ABB RAPID module: RRC_DataGlobal_Ctrl.sysx

MODULE RRC_DataGlobal_Ctrl(SYSMODULE)
    !***********************************************************************************
    !
    ! ETH Zurich / Robotic Fabrication Lab
    ! HIB C13 / Stefano-Franscini-Platz 1
    ! CH-8093 Zurich
    !
    !***********************************************************************************
    !
    ! PROJECT     :  RRC - Rapid Robot Communication
    !
    ! FUNCTION    :  Inclouds all project spezific global datas
    !
    ! AUTHOR      :  Philippe Fleischmann
    !
    ! EMAIL       :  rrc@arch.ethz.ch
    !
    ! HISTORY     :  2019.02.22
    !
    ! Copyright   :  ETH Zurich (CH) 2019
    !                - Philippe Fleischmann
    !                - Michael Lyrenmann
    !                - Gonzalo Casas
    !
    ! License     :  This code base is governed by an EULA (End-User License Agreement)
    !                which you have received together with the software.
    !                You are not allowed to use the software on a real robots
    !                without a signed EULA.
    !
    !                A copy of the EULA content is in the controller task (T_CTRL).
    !
    !***********************************************************************************

    !************************************************
    ! Declaration :     bool
    !************************************************
    !
    PERS bool b_RRC_TaskReceiverOn:=TRUE;
    PERS bool b_RRC_TaskSenderOn:=TRUE;
    !
    PERS bool b_RRC_CtrlWaitForJob:=TRUE;
    PERS bool b_RRC_CtrlHamModOn:=FALSE;
    PERS bool b_RRC_CtrlInUse:=FALSE;
    PERS bool b_RRC_AutoIPAddress:=FALSE;
    PERS bool b_RRC_VirtualCustomPorts:=FALSE;
    !
    ! Channels
    PERS bool b_RRC_Com{n_RRC_NumOfCha}:=[TRUE,FALSE,FALSE,FALSE];
    PERS bool b_RRC_SIDCheck{n_RRC_NumOfCha}:=[TRUE,FALSE,FALSE,FALSE];
    PERS bool b_RRC_SIDErrorStop{n_RRC_NumOfCha}:=[FALSE,FALSE,FALSE,FALSE];
    PERS bool b_RRC_LogPro{n_RRC_NumOfCha}:=[FALSE,FALSE,FALSE,FALSE];
    !
    ! Client information
    PERS bool b_RRC_PPMain:=TRUE;
    !
    ! Activate or deactivate a event log message
    PERS bool b_RRC_EvLogReadAndUnpackTime:=FALSE;
    PERS bool b_RRC_EvLogPackAndSendTime:=FALSE;
    PERS bool b_RRC_EvLogMsgInUntilMsgOutTime:=FALSE;
    !
    ! Temporary to measure the feedback loop
    PERS bool b_RRC_FeedbackOut:=TRUE;

    !************************************************
    ! Declaration :     num
    !************************************************
    !
    !* PERS num n_RRC_WritePtrSenBufRob1:=1;
    PERS num n_RRC_WritePtrSenBufCtrl{n_RRC_NumOfCha}:=[0,0,0,0];
    PERS num n_RRC_WritePtrSenBufRob{n_RRC_NumOfCha}:=[4,0,0,0];
    !* PERS num n_RRC_SIDMax:=8388608;
    PERS num n_RRC_SIDMax:=1000000;
    !
    PERS num n_RRC_R1_ChaNr:=1;
    PERS num n_RRC_R2_ChaNr:=2;
    PERS num n_RRC_R3_ChaNr:=3;
    PERS num n_RRC_R4_ChaNr:=4;
    !
    PERS num n_RRC_SocketPortRec{n_RRC_NumOfCha}:=[30101,30102,30103,30104];
    PERS num n_RRC_SocketPortSen{n_RRC_NumOfCha}:=[30201,30202,30203,30204];
    !
    PERS num n_RRC_TimeTaskLiAll:=0.1;
    PERS num n_RRC_TimeTPMsg:=0.5;
    !
    PERS num n_RRC_ProtocolVersion:=2;

    !************************************************
    ! Declaration :     string
    !************************************************
    !
    PERS string n_RRC_Version:="v1.1.0";
    !
    PERS string st_RRC_CurCtrlJob:="RRC";
    PERS string st_RRC_JobForCtrl:="r_A031_HamMod";
    !
    PERS string st_RRC_IP_Address:="192.168.125.1";
    PERS string st_RRC_IP_AddressVC:="127.0.0.1";
    PERS string st_RRC_IP_AddressMan:="192.168.125.1";
    !
    ! System data
    PERS string st_RRC_SerialNr:="15000-100220";
    PERS string st_RRC_SoftwareVersion:="7.7.1+296";
    PERS string st_RRC_RobotWare:="7.7.1";
    PERS string st_RRC_ControllerID:="15000-100220";
    PERS string st_RRC_WAN_IP:="0.0.0.0";
    PERS string st_RRC_ControllerLang:="en";
    PERS string st_RRC_SystemName:="15000-100220";

    !************************************************
    ! Declaration :     tasklist
    !************************************************
    !
    PERS tasks tl_RRC_All{7}:=[["T_CTRL"],["T_RX"],["T_TX"],["T_ROB1"],[""],[""],[""]];

    !************************************************
    ! Declaration :     syncident
    !************************************************
    !
    VAR syncident id_RRC_MainSta;
    VAR syncident id_RRC_MainEnd;
    !
    VAR syncident id_RRC_InitSta;
    VAR syncident id_RRC_InitCtrl;
    VAR syncident id_RRC_InitEnd;

    !************************************************
    ! Declaration :     RRC_Channel
    !************************************************
    !
    PERS RRC_Channel ch_RRC_Channels:=[["T_ROB1",1],["T_ROB2",2],["T_ROB3",3],["T_ROB4",4]];

    !************************************************
    ! Declaration :     RRC_buffer_msg
    !************************************************
    !
    ! Receiver buffer for controller
    PERS RRC_buffer_msg bm_RRC_RecBufferCtrl{n_RRC_NumOfCha,10}:=[
    [[[0,0,0,"",0,0,"",0,0,0,"",0,"",0,"",0,"",0,"",0,"",0,"",0,"",0,0,0,0,0,0,0,0,0,0,0,0,0,0,0,0,0,0,0,0,0,0,0,0,0,0,0,0,0,0,0,0,0,0,0,0,0],FALSE],
    [[0,0,0,"",0,0,"",0,0,0,"",0,"",0,"",0,"",0,"",0,"",0,"",0,"",0,0,0,0,0,0,0,0,0,0,0,0,0,0,0,0,0,0,0,0,0,0,0,0,0,0,0,0,0,0,0,0,0,0,0,0,0],FALSE],
    [[0,0,0,"",0,0,"",0,0,0,"",0,"",0,"",0,"",0,"",0,"",0,"",0,"",0,0,0,0,0,0,0,0,0,0,0,0,0,0,0,0,0,0,0,0,0,0,0,0,0,0,0,0,0,0,0,0,0,0,0,0,0],FALSE],
    [[0,0,0,"",0,0,"",0,0,0,"",0,"",0,"",0,"",0,"",0,"",0,"",0,"",0,0,0,0,0,0,0,0,0,0,0,0,0,0,0,0,0,0,0,0,0,0,0,0,0,0,0,0,0,0,0,0,0,0,0,0,0],FALSE],
    [[0,0,0,"",0,0,"",0,0,0,"",0,"",0,"",0,"",0,"",0,"",0,"",0,"",0,0,0,0,0,0,0,0,0,0,0,0,0,0,0,0,0,0,0,0,0,0,0,0,0,0,0,0,0,0,0,0,0,0,0,0,0],FALSE],
    [[0,0,0,"",0,0,"",0,0,0,"",0,"",0,"",0,"",0,"",0,"",0,"",0,"",0,0,0,0,0,0,0,0,0,0,0,0,0,0,0,0,0,0,0,0,0,0,0,0,0,0,0,0,0,0,0,0,0,0,0,0,0],FALSE],
    [[0,0,0,"",0,0,"",0,0,0,"",0,"",0,"",0,"",0,"",0,"",0,"",0,"",0,0,0,0,0,0,0,0,0,0,0,0,0,0,0,0,0,0,0,0,0,0,0,0,0,0,0,0,0,0,0,0,0,0,0,0,0],FALSE],
    [[0,0,0,"",0,0,"",0,0,0,"",0,"",0,"",0,"",0,"",0,"",0,"",0,"",0,0,0,0,0,0,0,0,0,0,0,0,0,0,0,0,0,0,0,0,0,0,0,0,0,0,0,0,0,0,0,0,0,0,0,0,0],FALSE],
    [[0,0,0,"",0,0,"",0,0,0,"",0,"",0,"",0,"",0,"",0,"",0,"",0,"",0,0,0,0,0,0,0,0,0,0,0,0,0,0,0,0,0,0,0,0,0,0,0,0,0,0,0,0,0,0,0,0,0,0,0,0,0],FALSE],
    [[0,0,0,"",0,0,"",0,0,0,"",0,"",0,"",0,"",0,"",0,"",0,"",0,"",0,0,0,0,0,0,0,0,0,0,0,0,0,0,0,0,0,0,0,0,0,0,0,0,0,0,0,0,0,0,0,0,0,0,0,0,0],FALSE]],

    [[[0,0,0,"",0,0,"",0,0,0,"",0,"",0,"",0,"",0,"",0,"",0,"",0,"",0,0,0,0,0,0,0,0,0,0,0,0,0,0,0,0,0,0,0,0,0,0,0,0,0,0,0,0,0,0,0,0,0,0,0,0,0],FALSE],
    [[0,0,0,"",0,0,"",0,0,0,"",0,"",0,"",0,"",0,"",0,"",0,"",0,"",0,0,0,0,0,0,0,0,0,0,0,0,0,0,0,0,0,0,0,0,0,0,0,0,0,0,0,0,0,0,0,0,0,0,0,0,0],FALSE],
    [[0,0,0,"",0,0,"",0,0,0,"",0,"",0,"",0,"",0,"",0,"",0,"",0,"",0,0,0,0,0,0,0,0,0,0,0,0,0,0,0,0,0,0,0,0,0,0,0,0,0,0,0,0,0,0,0,0,0,0,0,0,0],FALSE],
    [[0,0,0,"",0,0,"",0,0,0,"",0,"",0,"",0,"",0,"",0,"",0,"",0,"",0,0,0,0,0,0,0,0,0,0,0,0,0,0,0,0,0,0,0,0,0,0,0,0,0,0,0,0,0,0,0,0,0,0,0,0,0],FALSE],
    [[0,0,0,"",0,0,"",0,0,0,"",0,"",0,"",0,"",0,"",0,"",0,"",0,"",0,0,0,0,0,0,0,0,0,0,0,0,0,0,0,0,0,0,0,0,0,0,0,0,0,0,0,0,0,0,0,0,0,0,0,0,0],FALSE],
    [[0,0,0,"",0,0,"",0,0,0,"",0,"",0,"",0,"",0,"",0,"",0,"",0,"",0,0,0,0,0,0,0,0,0,0,0,0,0,0,0,0,0,0,0,0,0,0,0,0,0,0,0,0,0,0,0,0,0,0,0,0,0],FALSE],
    [[0,0,0,"",0,0,"",0,0,0,"",0,"",0,"",0,"",0,"",0,"",0,"",0,"",0,0,0,0,0,0,0,0,0,0,0,0,0,0,0,0,0,0,0,0,0,0,0,0,0,0,0,0,0,0,0,0,0,0,0,0,0],FALSE],
    [[0,0,0,"",0,0,"",0,0,0,"",0,"",0,"",0,"",0,"",0,"",0,"",0,"",0,0,0,0,0,0,0,0,0,0,0,0,0,0,0,0,0,0,0,0,0,0,0,0,0,0,0,0,0,0,0,0,0,0,0,0,0],FALSE],
    [[0,0,0,"",0,0,"",0,0,0,"",0,"",0,"",0,"",0,"",0,"",0,"",0,"",0,0,0,0,0,0,0,0,0,0,0,0,0,0,0,0,0,0,0,0,0,0,0,0,0,0,0,0,0,0,0,0,0,0,0,0,0],FALSE],
    [[0,0,0,"",0,0,"",0,0,0,"",0,"",0,"",0,"",0,"",0,"",0,"",0,"",0,0,0,0,0,0,0,0,0,0,0,0,0,0,0,0,0,0,0,0,0,0,0,0,0,0,0,0,0,0,0,0,0,0,0,0,0],FALSE]],

    [[[0,0,0,"",0,0,"",0,0,0,"",0,"",0,"",0,"",0,"",0,"",0,"",0,"",0,0,0,0,0,0,0,0,0,0,0,0,0,0,0,0,0,0,0,0,0,0,0,0,0,0,0,0,0,0,0,0,0,0,0,0,0],FALSE],
    [[0,0,0,"",0,0,"",0,0,0,"",0,"",0,"",0,"",0,"",0,"",0,"",0,"",0,0,0,0,0,0,0,0,0,0,0,0,0,0,0,0,0,0,0,0,0,0,0,0,0,0,0,0,0,0,0,0,0,0,0,0,0],FALSE],
    [[0,0,0,"",0,0,"",0,0,0,"",0,"",0,"",0,"",0,"",0,"",0,"",0,"",0,0,0,0,0,0,0,0,0,0,0,0,0,0,0,0,0,0,0,0,0,0,0,0,0,0,0,0,0,0,0,0,0,0,0,0,0],FALSE],
    [[0,0,0,"",0,0,"",0,0,0,"",0,"",0,"",0,"",0,"",0,"",0,"",0,"",0,0,0,0,0,0,0,0,0,0,0,0,0,0,0,0,0,0,0,0,0,0,0,0,0,0,0,0,0,0,0,0,0,0,0,0,0],FALSE],
    [[0,0,0,"",0,0,"",0,0,0,"",0,"",0,"",0,"",0,"",0,"",0,"",0,"",0,0,0,0,0,0,0,0,0,0,0,0,0,0,0,0,0,0,0,0,0,0,0,0,0,0,0,0,0,0,0,0,0,0,0,0,0],FALSE],
    [[0,0,0,"",0,0,"",0,0,0,"",0,"",0,"",0,"",0,"",0,"",0,"",0,"",0,0,0,0,0,0,0,0,0,0,0,0,0,0,0,0,0,0,0,0,0,0,0,0,0,0,0,0,0,0,0,0,0,0,0,0,0],FALSE],
    [[0,0,0,"",0,0,"",0,0,0,"",0,"",0,"",0,"",0,"",0,"",0,"",0,"",0,0,0,0,0,0,0,0,0,0,0,0,0,0,0,0,0,0,0,0,0,0,0,0,0,0,0,0,0,0,0,0,0,0,0,0,0],FALSE],
    [[0,0,0,"",0,0,"",0,0,0,"",0,"",0,"",0,"",0,"",0,"",0,"",0,"",0,0,0,0,0,0,0,0,0,0,0,0,0,0,0,0,0,0,0,0,0,0,0,0,0,0,0,0,0,0,0,0,0,0,0,0,0],FALSE],
    [[0,0,0,"",0,0,"",0,0,0,"",0,"",0,"",0,"",0,"",0,"",0,"",0,"",0,0,0,0,0,0,0,0,0,0,0,0,0,0,0,0,0,0,0,0,0,0,0,0,0,0,0,0,0,0,0,0,0,0,0,0,0],FALSE],
    [[0,0,0,"",0,0,"",0,0,0,"",0,"",0,"",0,"",0,"",0,"",0,"",0,"",0,0,0,0,0,0,0,0,0,0,0,0,0,0,0,0,0,0,0,0,0,0,0,0,0,0,0,0,0,0,0,0,0,0,0,0,0],FALSE]],

    [[[0,0,0,"",0,0,"",0,0,0,"",0,"",0,"",0,"",0,"",0,"",0,"",0,"",0,0,0,0,0,0,0,0,0,0,0,0,0,0,0,0,0,0,0,0,0,0,0,0,0,0,0,0,0,0,0,0,0,0,0,0,0],FALSE],
    [[0,0,0,"",0,0,"",0,0,0,"",0,"",0,"",0,"",0,"",0,"",0,"",0,"",0,0,0,0,0,0,0,0,0,0,0,0,0,0,0,0,0,0,0,0,0,0,0,0,0,0,0,0,0,0,0,0,0,0,0,0,0],FALSE],
    [[0,0,0,"",0,0,"",0,0,0,"",0,"",0,"",0,"",0,"",0,"",0,"",0,"",0,0,0,0,0,0,0,0,0,0,0,0,0,0,0,0,0,0,0,0,0,0,0,0,0,0,0,0,0,0,0,0,0,0,0,0,0],FALSE],
    [[0,0,0,"",0,0,"",0,0,0,"",0,"",0,"",0,"",0,"",0,"",0,"",0,"",0,0,0,0,0,0,0,0,0,0,0,0,0,0,0,0,0,0,0,0,0,0,0,0,0,0,0,0,0,0,0,0,0,0,0,0,0],FALSE],
    [[0,0,0,"",0,0,"",0,0,0,"",0,"",0,"",0,"",0,"",0,"",0,"",0,"",0,0,0,0,0,0,0,0,0,0,0,0,0,0,0,0,0,0,0,0,0,0,0,0,0,0,0,0,0,0,0,0,0,0,0,0,0],FALSE],
    [[0,0,0,"",0,0,"",0,0,0,"",0,"",0,"",0,"",0,"",0,"",0,"",0,"",0,0,0,0,0,0,0,0,0,0,0,0,0,0,0,0,0,0,0,0,0,0,0,0,0,0,0,0,0,0,0,0,0,0,0,0,0],FALSE],
    [[0,0,0,"",0,0,"",0,0,0,"",0,"",0,"",0,"",0,"",0,"",0,"",0,"",0,0,0,0,0,0,0,0,0,0,0,0,0,0,0,0,0,0,0,0,0,0,0,0,0,0,0,0,0,0,0,0,0,0,0,0,0],FALSE],
    [[0,0,0,"",0,0,"",0,0,0,"",0,"",0,"",0,"",0,"",0,"",0,"",0,"",0,0,0,0,0,0,0,0,0,0,0,0,0,0,0,0,0,0,0,0,0,0,0,0,0,0,0,0,0,0,0,0,0,0,0,0,0],FALSE],
    [[0,0,0,"",0,0,"",0,0,0,"",0,"",0,"",0,"",0,"",0,"",0,"",0,"",0,0,0,0,0,0,0,0,0,0,0,0,0,0,0,0,0,0,0,0,0,0,0,0,0,0,0,0,0,0,0,0,0,0,0,0,0],FALSE],
    [[0,0,0,"",0,0,"",0,0,0,"",0,"",0,"",0,"",0,"",0,"",0,"",0,"",0,0,0,0,0,0,0,0,0,0,0,0,0,0,0,0,0,0,0,0,0,0,0,0,0,0,0,0,0,0,0,0,0,0,0,0,0],FALSE]]];

    !
    ! Receiver buffer for robots
    PERS RRC_buffer_msg bm_RRC_RecBufferRob{n_RRC_NumOfCha,10}:=[
    [[[5,0,12,"r_RRC_MoveTo",1,0,"",0,1,6,"FrameL",0,"",0,"",0,"",0,"",0,"",0,"",0,"",15,0.00865957,478.991,218.552,7.09225E-05,0.923882,-0.382677,3.67571E-05,0,0,0,0,0,0,300,-1,0,0,0,0,0,0,0,0,0,0,0,0,0,0,0,0,0,0,0,0,0],FALSE],
    [[6,0,12,"r_RRC_MoveTo",1,0,"",0,1,6,"FrameL",0,"",0,"",0,"",0,"",0,"",0,"",0,"",15,550.001,-0.000425997,717.995,-1.78564E-06,-0.382682,0.92388,7.29413E-07,0,0,0,0,0,0,300,-1,0,0,0,0,0,0,0,0,0,0,0,0,0,0,0,0,0,0,0,0,0],FALSE],
    [[7,0,12,"r_RRC_MoveTo",1,0,"",0,1,6,"FrameL",0,"",0,"",0,"",0,"",0,"",0,"",0,"",15,697.669,-21.8245,303.5,0,-0.320157,0.947365,0,0,0,0,0,0,0,300,-1,0,0,0,0,0,0,0,0,0,0,0,0,0,0,0,0,0,0,0,0,0],FALSE],
    [[8,0,12,"r_RRC_MoveTo",1,0,"",0,1,6,"FrameL",0,"",0,"",0,"",0,"",0,"",0,"",0,"",15,697.669,-21.8245,253.5,0,-0.320157,0.947365,0,0,0,0,0,0,0,300,-1,0,0,0,0,0,0,0,0,0,0,0,0,0,0,0,0,0,0,0,0,0],FALSE],
    [[9,0,16,"r_RRC_SetDigital",0,0,"",0,1,22,"ABB_Scalable_IO_0_DO16",0,"",0,"",0,"",0,"",0,"",0,"",0,"",1,1,-21.8245,253.5,0,-0.320157,0.947365,0,0,0,0,0,0,0,300,-1,0,0,0,0,0,0,0,0,0,0,0,0,0,0,0,0,0,0,0,0,0],FALSE],
    [[10,0,12,"r_RRC_MoveTo",1,0,"",0,1,6,"FrameL",0,"",0,"",0,"",0,"",0,"",0,"",0,"",15,697.669,-21.8245,303.5,0,-0.320157,0.947365,0,0,0,0,0,0,0,300,-1,0,0,0,0,0,0,0,0,0,0,0,0,0,0,0,0,0,0,0,0,0],FALSE],
    [[11,0,12,"r_RRC_MoveTo",1,0,"",0,1,6,"FrameL",0,"",0,"",0,"",0,"",0,"",0,"",0,"",15,550.001,-0.000425997,717.995,-1.78564E-06,-0.382682,0.92388,7.29413E-07,0,0,0,0,0,0,300,-1,0,0,0,0,0,0,0,0,0,0,0,0,0,0,0,0,0,0,0,0,0],FALSE],
    [[12,0,12,"r_RRC_MoveTo",1,0,"",0,1,6,"FrameL",0,"",0,"",0,"",0,"",0,"",0,"",0,"",15,0.00865957,478.991,218.552,7.09225E-05,0.923882,-0.382677,3.67571E-05,0,0,0,0,0,0,300,-1,0,0,0,0,0,0,0,0,0,0,0,0,0,0,0,0,0,0,0,0,0],FALSE],
    [[13,0,12,"r_RRC_MoveTo",1,0,"",0,1,6,"FrameL",0,"",0,"",0,"",0,"",0,"",0,"",0,"",15,0.00865957,478.991,168.552,7.09225E-05,0.923882,-0.382677,3.67571E-05,0,0,0,0,0,0,300,-1,0,0,0,0,0,0,0,0,0,0,0,0,0,0,0,0,0,0,0,0,0],FALSE],
    [[4,0,14,"r_RRC_WaitTime",1,0,"",0,0,22,"ABB_Scalable_IO_0_DO16",0,"",0,"",0,"",0,"",0,"",0,"",0,"",1,1,478.991,168.552,7.09225E-05,0.923882,-0.382677,3.67571E-05,0,0,0,0,0,0,300,-1,0,0,0,0,0,0,0,0,0,0,0,0,0,0,0,0,0,0,0,0,0],FALSE]],

    [[[0,0,0,"",0,0,"",0,0,0,"",0,"",0,"",0,"",0,"",0,"",0,"",0,"",0,0,0,0,0,0,0,0,0,0,0,0,0,0,0,0,0,0,0,0,0,0,0,0,0,0,0,0,0,0,0,0,0,0,0,0,0],FALSE],
    [[0,0,0,"",0,0,"",0,0,0,"",0,"",0,"",0,"",0,"",0,"",0,"",0,"",0,0,0,0,0,0,0,0,0,0,0,0,0,0,0,0,0,0,0,0,0,0,0,0,0,0,0,0,0,0,0,0,0,0,0,0,0],FALSE],
    [[0,0,0,"",0,0,"",0,0,0,"",0,"",0,"",0,"",0,"",0,"",0,"",0,"",0,0,0,0,0,0,0,0,0,0,0,0,0,0,0,0,0,0,0,0,0,0,0,0,0,0,0,0,0,0,0,0,0,0,0,0,0],FALSE],
    [[0,0,0,"",0,0,"",0,0,0,"",0,"",0,"",0,"",0,"",0,"",0,"",0,"",0,0,0,0,0,0,0,0,0,0,0,0,0,0,0,0,0,0,0,0,0,0,0,0,0,0,0,0,0,0,0,0,0,0,0,0,0],FALSE],
    [[0,0,0,"",0,0,"",0,0,0,"",0,"",0,"",0,"",0,"",0,"",0,"",0,"",0,0,0,0,0,0,0,0,0,0,0,0,0,0,0,0,0,0,0,0,0,0,0,0,0,0,0,0,0,0,0,0,0,0,0,0,0],FALSE],
    [[0,0,0,"",0,0,"",0,0,0,"",0,"",0,"",0,"",0,"",0,"",0,"",0,"",0,0,0,0,0,0,0,0,0,0,0,0,0,0,0,0,0,0,0,0,0,0,0,0,0,0,0,0,0,0,0,0,0,0,0,0,0],FALSE],
    [[0,0,0,"",0,0,"",0,0,0,"",0,"",0,"",0,"",0,"",0,"",0,"",0,"",0,0,0,0,0,0,0,0,0,0,0,0,0,0,0,0,0,0,0,0,0,0,0,0,0,0,0,0,0,0,0,0,0,0,0,0,0],FALSE],
    [[0,0,0,"",0,0,"",0,0,0,"",0,"",0,"",0,"",0,"",0,"",0,"",0,"",0,0,0,0,0,0,0,0,0,0,0,0,0,0,0,0,0,0,0,0,0,0,0,0,0,0,0,0,0,0,0,0,0,0,0,0,0],FALSE],
    [[0,0,0,"",0,0,"",0,0,0,"",0,"",0,"",0,"",0,"",0,"",0,"",0,"",0,0,0,0,0,0,0,0,0,0,0,0,0,0,0,0,0,0,0,0,0,0,0,0,0,0,0,0,0,0,0,0,0,0,0,0,0],FALSE],
    [[0,0,0,"",0,0,"",0,0,0,"",0,"",0,"",0,"",0,"",0,"",0,"",0,"",0,0,0,0,0,0,0,0,0,0,0,0,0,0,0,0,0,0,0,0,0,0,0,0,0,0,0,0,0,0,0,0,0,0,0,0,0],FALSE]],

    [[[0,0,0,"",0,0,"",0,0,0,"",0,"",0,"",0,"",0,"",0,"",0,"",0,"",0,0,0,0,0,0,0,0,0,0,0,0,0,0,0,0,0,0,0,0,0,0,0,0,0,0,0,0,0,0,0,0,0,0,0,0,0],FALSE],
    [[0,0,0,"",0,0,"",0,0,0,"",0,"",0,"",0,"",0,"",0,"",0,"",0,"",0,0,0,0,0,0,0,0,0,0,0,0,0,0,0,0,0,0,0,0,0,0,0,0,0,0,0,0,0,0,0,0,0,0,0,0,0],FALSE],
    [[0,0,0,"",0,0,"",0,0,0,"",0,"",0,"",0,"",0,"",0,"",0,"",0,"",0,0,0,0,0,0,0,0,0,0,0,0,0,0,0,0,0,0,0,0,0,0,0,0,0,0,0,0,0,0,0,0,0,0,0,0,0],FALSE],
    [[0,0,0,"",0,0,"",0,0,0,"",0,"",0,"",0,"",0,"",0,"",0,"",0,"",0,0,0,0,0,0,0,0,0,0,0,0,0,0,0,0,0,0,0,0,0,0,0,0,0,0,0,0,0,0,0,0,0,0,0,0,0],FALSE],
    [[0,0,0,"",0,0,"",0,0,0,"",0,"",0,"",0,"",0,"",0,"",0,"",0,"",0,0,0,0,0,0,0,0,0,0,0,0,0,0,0,0,0,0,0,0,0,0,0,0,0,0,0,0,0,0,0,0,0,0,0,0,0],FALSE],
    [[0,0,0,"",0,0,"",0,0,0,"",0,"",0,"",0,"",0,"",0,"",0,"",0,"",0,0,0,0,0,0,0,0,0,0,0,0,0,0,0,0,0,0,0,0,0,0,0,0,0,0,0,0,0,0,0,0,0,0,0,0,0],FALSE],
    [[0,0,0,"",0,0,"",0,0,0,"",0,"",0,"",0,"",0,"",0,"",0,"",0,"",0,0,0,0,0,0,0,0,0,0,0,0,0,0,0,0,0,0,0,0,0,0,0,0,0,0,0,0,0,0,0,0,0,0,0,0,0],FALSE],
    [[0,0,0,"",0,0,"",0,0,0,"",0,"",0,"",0,"",0,"",0,"",0,"",0,"",0,0,0,0,0,0,0,0,0,0,0,0,0,0,0,0,0,0,0,0,0,0,0,0,0,0,0,0,0,0,0,0,0,0,0,0,0],FALSE],
    [[0,0,0,"",0,0,"",0,0,0,"",0,"",0,"",0,"",0,"",0,"",0,"",0,"",0,0,0,0,0,0,0,0,0,0,0,0,0,0,0,0,0,0,0,0,0,0,0,0,0,0,0,0,0,0,0,0,0,0,0,0,0],FALSE],
    [[0,0,0,"",0,0,"",0,0,0,"",0,"",0,"",0,"",0,"",0,"",0,"",0,"",0,0,0,0,0,0,0,0,0,0,0,0,0,0,0,0,0,0,0,0,0,0,0,0,0,0,0,0,0,0,0,0,0,0,0,0,0],FALSE]],

    [[[0,0,0,"",0,0,"",0,0,0,"",0,"",0,"",0,"",0,"",0,"",0,"",0,"",0,0,0,0,0,0,0,0,0,0,0,0,0,0,0,0,0,0,0,0,0,0,0,0,0,0,0,0,0,0,0,0,0,0,0,0,0],FALSE],
    [[0,0,0,"",0,0,"",0,0,0,"",0,"",0,"",0,"",0,"",0,"",0,"",0,"",0,0,0,0,0,0,0,0,0,0,0,0,0,0,0,0,0,0,0,0,0,0,0,0,0,0,0,0,0,0,0,0,0,0,0,0,0],FALSE],
    [[0,0,0,"",0,0,"",0,0,0,"",0,"",0,"",0,"",0,"",0,"",0,"",0,"",0,0,0,0,0,0,0,0,0,0,0,0,0,0,0,0,0,0,0,0,0,0,0,0,0,0,0,0,0,0,0,0,0,0,0,0,0],FALSE],
    [[0,0,0,"",0,0,"",0,0,0,"",0,"",0,"",0,"",0,"",0,"",0,"",0,"",0,0,0,0,0,0,0,0,0,0,0,0,0,0,0,0,0,0,0,0,0,0,0,0,0,0,0,0,0,0,0,0,0,0,0,0,0],FALSE],
    [[0,0,0,"",0,0,"",0,0,0,"",0,"",0,"",0,"",0,"",0,"",0,"",0,"",0,0,0,0,0,0,0,0,0,0,0,0,0,0,0,0,0,0,0,0,0,0,0,0,0,0,0,0,0,0,0,0,0,0,0,0,0],FALSE],
    [[0,0,0,"",0,0,"",0,0,0,"",0,"",0,"",0,"",0,"",0,"",0,"",0,"",0,0,0,0,0,0,0,0,0,0,0,0,0,0,0,0,0,0,0,0,0,0,0,0,0,0,0,0,0,0,0,0,0,0,0,0,0],FALSE],
    [[0,0,0,"",0,0,"",0,0,0,"",0,"",0,"",0,"",0,"",0,"",0,"",0,"",0,0,0,0,0,0,0,0,0,0,0,0,0,0,0,0,0,0,0,0,0,0,0,0,0,0,0,0,0,0,0,0,0,0,0,0,0],FALSE],
    [[0,0,0,"",0,0,"",0,0,0,"",0,"",0,"",0,"",0,"",0,"",0,"",0,"",0,0,0,0,0,0,0,0,0,0,0,0,0,0,0,0,0,0,0,0,0,0,0,0,0,0,0,0,0,0,0,0,0,0,0,0,0],FALSE],
    [[0,0,0,"",0,0,"",0,0,0,"",0,"",0,"",0,"",0,"",0,"",0,"",0,"",0,0,0,0,0,0,0,0,0,0,0,0,0,0,0,0,0,0,0,0,0,0,0,0,0,0,0,0,0,0,0,0,0,0,0,0,0],FALSE],
    [[0,0,0,"",0,0,"",0,0,0,"",0,"",0,"",0,"",0,"",0,"",0,"",0,"",0,0,0,0,0,0,0,0,0,0,0,0,0,0,0,0,0,0,0,0,0,0,0,0,0,0,0,0,0,0,0,0,0,0,0,0,0],FALSE]]];

    !
    ! Sender buffer for controller
    PERS RRC_buffer_msg bm_RRC_SenBufferCtrl{n_RRC_NumOfCha,10}:=[
    [[[0,0,0,"",0,0,"",0,0,0,"",0,"",0,"",0,"",0,"",0,"",0,"",0,"",0,0,0,0,0,0,0,0,0,0,0,0,0,0,0,0,0,0,0,0,0,0,0,0,0,0,0,0,0,0,0,0,0,0,0,0,0],FALSE],
    [[0,0,0,"",0,0,"",0,0,0,"",0,"",0,"",0,"",0,"",0,"",0,"",0,"",0,0,0,0,0,0,0,0,0,0,0,0,0,0,0,0,0,0,0,0,0,0,0,0,0,0,0,0,0,0,0,0,0,0,0,0,0],FALSE],
    [[0,0,0,"",0,0,"",0,0,0,"",0,"",0,"",0,"",0,"",0,"",0,"",0,"",0,0,0,0,0,0,0,0,0,0,0,0,0,0,0,0,0,0,0,0,0,0,0,0,0,0,0,0,0,0,0,0,0,0,0,0,0],FALSE],
    [[0,0,0,"",0,0,"",0,0,0,"",0,"",0,"",0,"",0,"",0,"",0,"",0,"",0,0,0,0,0,0,0,0,0,0,0,0,0,0,0,0,0,0,0,0,0,0,0,0,0,0,0,0,0,0,0,0,0,0,0,0,0],FALSE],
    [[0,0,0,"",0,0,"",0,0,0,"",0,"",0,"",0,"",0,"",0,"",0,"",0,"",0,0,0,0,0,0,0,0,0,0,0,0,0,0,0,0,0,0,0,0,0,0,0,0,0,0,0,0,0,0,0,0,0,0,0,0,0],FALSE],
    [[0,0,0,"",0,0,"",0,0,0,"",0,"",0,"",0,"",0,"",0,"",0,"",0,"",0,0,0,0,0,0,0,0,0,0,0,0,0,0,0,0,0,0,0,0,0,0,0,0,0,0,0,0,0,0,0,0,0,0,0,0,0],FALSE],
    [[0,0,0,"",0,0,"",0,0,0,"",0,"",0,"",0,"",0,"",0,"",0,"",0,"",0,0,0,0,0,0,0,0,0,0,0,0,0,0,0,0,0,0,0,0,0,0,0,0,0,0,0,0,0,0,0,0,0,0,0,0,0],FALSE],
    [[0,0,0,"",0,0,"",0,0,0,"",0,"",0,"",0,"",0,"",0,"",0,"",0,"",0,0,0,0,0,0,0,0,0,0,0,0,0,0,0,0,0,0,0,0,0,0,0,0,0,0,0,0,0,0,0,0,0,0,0,0,0],FALSE],
    [[0,0,0,"",0,0,"",0,0,0,"",0,"",0,"",0,"",0,"",0,"",0,"",0,"",0,0,0,0,0,0,0,0,0,0,0,0,0,0,0,0,0,0,0,0,0,0,0,0,0,0,0,0,0,0,0,0,0,0,0,0,0],FALSE],
    [[0,0,0,"",0,0,"",0,0,0,"",0,"",0,"",0,"",0,"",0,"",0,"",0,"",0,0,0,0,0,0,0,0,0,0,0,0,0,0,0,0,0,0,0,0,0,0,0,0,0,0,0,0,0,0,0,0,0,0,0,0,0],FALSE]],

    [[[0,0,0,"",0,0,"",0,0,0,"",0,"",0,"",0,"",0,"",0,"",0,"",0,"",0,0,0,0,0,0,0,0,0,0,0,0,0,0,0,0,0,0,0,0,0,0,0,0,0,0,0,0,0,0,0,0,0,0,0,0,0],FALSE],
    [[0,0,0,"",0,0,"",0,0,0,"",0,"",0,"",0,"",0,"",0,"",0,"",0,"",0,0,0,0,0,0,0,0,0,0,0,0,0,0,0,0,0,0,0,0,0,0,0,0,0,0,0,0,0,0,0,0,0,0,0,0,0],FALSE],
    [[0,0,0,"",0,0,"",0,0,0,"",0,"",0,"",0,"",0,"",0,"",0,"",0,"",0,0,0,0,0,0,0,0,0,0,0,0,0,0,0,0,0,0,0,0,0,0,0,0,0,0,0,0,0,0,0,0,0,0,0,0,0],FALSE],
    [[0,0,0,"",0,0,"",0,0,0,"",0,"",0,"",0,"",0,"",0,"",0,"",0,"",0,0,0,0,0,0,0,0,0,0,0,0,0,0,0,0,0,0,0,0,0,0,0,0,0,0,0,0,0,0,0,0,0,0,0,0,0],FALSE],
    [[0,0,0,"",0,0,"",0,0,0,"",0,"",0,"",0,"",0,"",0,"",0,"",0,"",0,0,0,0,0,0,0,0,0,0,0,0,0,0,0,0,0,0,0,0,0,0,0,0,0,0,0,0,0,0,0,0,0,0,0,0,0],FALSE],
    [[0,0,0,"",0,0,"",0,0,0,"",0,"",0,"",0,"",0,"",0,"",0,"",0,"",0,0,0,0,0,0,0,0,0,0,0,0,0,0,0,0,0,0,0,0,0,0,0,0,0,0,0,0,0,0,0,0,0,0,0,0,0],FALSE],
    [[0,0,0,"",0,0,"",0,0,0,"",0,"",0,"",0,"",0,"",0,"",0,"",0,"",0,0,0,0,0,0,0,0,0,0,0,0,0,0,0,0,0,0,0,0,0,0,0,0,0,0,0,0,0,0,0,0,0,0,0,0,0],FALSE],
    [[0,0,0,"",0,0,"",0,0,0,"",0,"",0,"",0,"",0,"",0,"",0,"",0,"",0,0,0,0,0,0,0,0,0,0,0,0,0,0,0,0,0,0,0,0,0,0,0,0,0,0,0,0,0,0,0,0,0,0,0,0,0],FALSE],
    [[0,0,0,"",0,0,"",0,0,0,"",0,"",0,"",0,"",0,"",0,"",0,"",0,"",0,0,0,0,0,0,0,0,0,0,0,0,0,0,0,0,0,0,0,0,0,0,0,0,0,0,0,0,0,0,0,0,0,0,0,0,0],FALSE],
    [[0,0,0,"",0,0,"",0,0,0,"",0,"",0,"",0,"",0,"",0,"",0,"",0,"",0,0,0,0,0,0,0,0,0,0,0,0,0,0,0,0,0,0,0,0,0,0,0,0,0,0,0,0,0,0,0,0,0,0,0,0,0],FALSE]],

    [[[0,0,0,"",0,0,"",0,0,0,"",0,"",0,"",0,"",0,"",0,"",0,"",0,"",0,0,0,0,0,0,0,0,0,0,0,0,0,0,0,0,0,0,0,0,0,0,0,0,0,0,0,0,0,0,0,0,0,0,0,0,0],FALSE],
    [[0,0,0,"",0,0,"",0,0,0,"",0,"",0,"",0,"",0,"",0,"",0,"",0,"",0,0,0,0,0,0,0,0,0,0,0,0,0,0,0,0,0,0,0,0,0,0,0,0,0,0,0,0,0,0,0,0,0,0,0,0,0],FALSE],
    [[0,0,0,"",0,0,"",0,0,0,"",0,"",0,"",0,"",0,"",0,"",0,"",0,"",0,0,0,0,0,0,0,0,0,0,0,0,0,0,0,0,0,0,0,0,0,0,0,0,0,0,0,0,0,0,0,0,0,0,0,0,0],FALSE],
    [[0,0,0,"",0,0,"",0,0,0,"",0,"",0,"",0,"",0,"",0,"",0,"",0,"",0,0,0,0,0,0,0,0,0,0,0,0,0,0,0,0,0,0,0,0,0,0,0,0,0,0,0,0,0,0,0,0,0,0,0,0,0],FALSE],
    [[0,0,0,"",0,0,"",0,0,0,"",0,"",0,"",0,"",0,"",0,"",0,"",0,"",0,0,0,0,0,0,0,0,0,0,0,0,0,0,0,0,0,0,0,0,0,0,0,0,0,0,0,0,0,0,0,0,0,0,0,0,0],FALSE],
    [[0,0,0,"",0,0,"",0,0,0,"",0,"",0,"",0,"",0,"",0,"",0,"",0,"",0,0,0,0,0,0,0,0,0,0,0,0,0,0,0,0,0,0,0,0,0,0,0,0,0,0,0,0,0,0,0,0,0,0,0,0,0],FALSE],
    [[0,0,0,"",0,0,"",0,0,0,"",0,"",0,"",0,"",0,"",0,"",0,"",0,"",0,0,0,0,0,0,0,0,0,0,0,0,0,0,0,0,0,0,0,0,0,0,0,0,0,0,0,0,0,0,0,0,0,0,0,0,0],FALSE],
    [[0,0,0,"",0,0,"",0,0,0,"",0,"",0,"",0,"",0,"",0,"",0,"",0,"",0,0,0,0,0,0,0,0,0,0,0,0,0,0,0,0,0,0,0,0,0,0,0,0,0,0,0,0,0,0,0,0,0,0,0,0,0],FALSE],
    [[0,0,0,"",0,0,"",0,0,0,"",0,"",0,"",0,"",0,"",0,"",0,"",0,"",0,0,0,0,0,0,0,0,0,0,0,0,0,0,0,0,0,0,0,0,0,0,0,0,0,0,0,0,0,0,0,0,0,0,0,0,0],FALSE],
    [[0,0,0,"",0,0,"",0,0,0,"",0,"",0,"",0,"",0,"",0,"",0,"",0,"",0,0,0,0,0,0,0,0,0,0,0,0,0,0,0,0,0,0,0,0,0,0,0,0,0,0,0,0,0,0,0,0,0,0,0,0,0],FALSE]],

    [[[0,0,0,"",0,0,"",0,0,0,"",0,"",0,"",0,"",0,"",0,"",0,"",0,"",0,0,0,0,0,0,0,0,0,0,0,0,0,0,0,0,0,0,0,0,0,0,0,0,0,0,0,0,0,0,0,0,0,0,0,0,0],FALSE],
    [[0,0,0,"",0,0,"",0,0,0,"",0,"",0,"",0,"",0,"",0,"",0,"",0,"",0,0,0,0,0,0,0,0,0,0,0,0,0,0,0,0,0,0,0,0,0,0,0,0,0,0,0,0,0,0,0,0,0,0,0,0,0],FALSE],
    [[0,0,0,"",0,0,"",0,0,0,"",0,"",0,"",0,"",0,"",0,"",0,"",0,"",0,0,0,0,0,0,0,0,0,0,0,0,0,0,0,0,0,0,0,0,0,0,0,0,0,0,0,0,0,0,0,0,0,0,0,0,0],FALSE],
    [[0,0,0,"",0,0,"",0,0,0,"",0,"",0,"",0,"",0,"",0,"",0,"",0,"",0,0,0,0,0,0,0,0,0,0,0,0,0,0,0,0,0,0,0,0,0,0,0,0,0,0,0,0,0,0,0,0,0,0,0,0,0],FALSE],
    [[0,0,0,"",0,0,"",0,0,0,"",0,"",0,"",0,"",0,"",0,"",0,"",0,"",0,0,0,0,0,0,0,0,0,0,0,0,0,0,0,0,0,0,0,0,0,0,0,0,0,0,0,0,0,0,0,0,0,0,0,0,0],FALSE],
    [[0,0,0,"",0,0,"",0,0,0,"",0,"",0,"",0,"",0,"",0,"",0,"",0,"",0,0,0,0,0,0,0,0,0,0,0,0,0,0,0,0,0,0,0,0,0,0,0,0,0,0,0,0,0,0,0,0,0,0,0,0,0],FALSE],
    [[0,0,0,"",0,0,"",0,0,0,"",0,"",0,"",0,"",0,"",0,"",0,"",0,"",0,0,0,0,0,0,0,0,0,0,0,0,0,0,0,0,0,0,0,0,0,0,0,0,0,0,0,0,0,0,0,0,0,0,0,0,0],FALSE],
    [[0,0,0,"",0,0,"",0,0,0,"",0,"",0,"",0,"",0,"",0,"",0,"",0,"",0,0,0,0,0,0,0,0,0,0,0,0,0,0,0,0,0,0,0,0,0,0,0,0,0,0,0,0,0,0,0,0,0,0,0,0,0],FALSE],
    [[0,0,0,"",0,0,"",0,0,0,"",0,"",0,"",0,"",0,"",0,"",0,"",0,"",0,0,0,0,0,0,0,0,0,0,0,0,0,0,0,0,0,0,0,0,0,0,0,0,0,0,0,0,0,0,0,0,0,0,0,0,0],FALSE],
    [[0,0,0,"",0,0,"",0,0,0,"",0,"",0,"",0,"",0,"",0,"",0,"",0,"",0,0,0,0,0,0,0,0,0,0,0,0,0,0,0,0,0,0,0,0,0,0,0,0,0,0,0,0,0,0,0,0,0,0,0,0,0],FALSE]]];

    !
    ! Sender buffer for robots
    PERS RRC_buffer_msg bm_RRC_SenBufferRob{n_RRC_NumOfCha,10}:=[
    [[[0,0,0,"r_RRC_MoveTo",0,0,"Done",10,0,0,"",0,"",0,"",0,"",0,"",0,"",0,"",0,"",0,0,0,0,0,0,0,0,0,0,0,0,0,0,0,0,0,0,0,0,0,0,0,0,0,0,0,0,0,0,0,0,0,0,0,0,0],FALSE],
    [[0,0,0,"r_RRC_MoveTo",0,0,"Done",11,0,0,"",0,"",0,"",0,"",0,"",0,"",0,"",0,"",0,0,0,0,0,0,0,0,0,0,0,0,0,0,0,0,0,0,0,0,0,0,0,0,0,0,0,0,0,0,0,0,0,0,0,0,0],FALSE],
    [[0,0,0,"r_RRC_MoveTo",0,0,"Done",12,0,0,"",0,"",0,"",0,"",0,"",0,"",0,"",0,"",0,0,0,0,0,0,0,0,0,0,0,0,0,0,0,0,0,0,0,0,0,0,0,0,0,0,0,0,0,0,0,0,0,0,0,0,0],FALSE],
    [[0,0,0,"r_RRC_MoveTo",0,0,"Done",13,0,0,"",0,"",0,"",0,"",0,"",0,"",0,"",0,"",0,0,0,0,0,0,0,0,0,0,0,0,0,0,0,0,0,0,0,0,0,0,0,0,0,0,0,0,0,0,0,0,0,0,0,0,0],FALSE],
    [[0,0,0,"r_RRC_MoveTo",0,0,"Done",13,0,0,"",0,"",0,"",0,"",0,"",0,"",0,"",0,"",0,0,0,0,0,0,0,0,0,0,0,0,0,0,0,0,0,0,0,0,0,0,0,0,0,0,0,0,0,0,0,0,0,0,0,0,0],FALSE],
    [[0,0,0,"r_RRC_WaitTime",0,0,"Done",4,0,0,"",0,"",0,"",0,"",0,"",0,"",0,"",0,"",0,0,0,0,0,0,0,0,0,0,0,0,0,0,0,0,0,0,0,0,0,0,0,0,0,0,0,0,0,0,0,0,0,0,0,0,0],FALSE],
    [[0,0,0,"r_RRC_MoveTo",0,0,"Done",5,0,0,"",0,"",0,"",0,"",0,"",0,"",0,"",0,"",0,0,0,0,0,0,0,0,0,0,0,0,0,0,0,0,0,0,0,0,0,0,0,0,0,0,0,0,0,0,0,0,0,0,0,0,0],FALSE],
    [[0,0,0,"r_RRC_MoveTo",0,0,"Done",6,0,0,"",0,"",0,"",0,"",0,"",0,"",0,"",0,"",0,0,0,0,0,0,0,0,0,0,0,0,0,0,0,0,0,0,0,0,0,0,0,0,0,0,0,0,0,0,0,0,0,0,0,0,0],FALSE],
    [[0,0,0,"r_RRC_MoveTo",0,0,"Done",7,0,0,"",0,"",0,"",0,"",0,"",0,"",0,"",0,"",0,0,0,0,0,0,0,0,0,0,0,0,0,0,0,0,0,0,0,0,0,0,0,0,0,0,0,0,0,0,0,0,0,0,0,0,0],FALSE],
    [[0,0,0,"r_RRC_MoveTo",0,0,"Done",8,0,0,"",0,"",0,"",0,"",0,"",0,"",0,"",0,"",0,0,0,0,0,0,0,0,0,0,0,0,0,0,0,0,0,0,0,0,0,0,0,0,0,0,0,0,0,0,0,0,0,0,0,0,0],FALSE]],

    [[[0,0,0,"",0,0,"",0,0,0,"",0,"",0,"",0,"",0,"",0,"",0,"",0,"",0,0,0,0,0,0,0,0,0,0,0,0,0,0,0,0,0,0,0,0,0,0,0,0,0,0,0,0,0,0,0,0,0,0,0,0,0],FALSE],
    [[0,0,0,"",0,0,"",0,0,0,"",0,"",0,"",0,"",0,"",0,"",0,"",0,"",0,0,0,0,0,0,0,0,0,0,0,0,0,0,0,0,0,0,0,0,0,0,0,0,0,0,0,0,0,0,0,0,0,0,0,0,0],FALSE],
    [[0,0,0,"",0,0,"",0,0,0,"",0,"",0,"",0,"",0,"",0,"",0,"",0,"",0,0,0,0,0,0,0,0,0,0,0,0,0,0,0,0,0,0,0,0,0,0,0,0,0,0,0,0,0,0,0,0,0,0,0,0,0],FALSE],
    [[0,0,0,"",0,0,"",0,0,0,"",0,"",0,"",0,"",0,"",0,"",0,"",0,"",0,0,0,0,0,0,0,0,0,0,0,0,0,0,0,0,0,0,0,0,0,0,0,0,0,0,0,0,0,0,0,0,0,0,0,0,0],FALSE],
    [[0,0,0,"",0,0,"",0,0,0,"",0,"",0,"",0,"",0,"",0,"",0,"",0,"",0,0,0,0,0,0,0,0,0,0,0,0,0,0,0,0,0,0,0,0,0,0,0,0,0,0,0,0,0,0,0,0,0,0,0,0,0],FALSE],
    [[0,0,0,"",0,0,"",0,0,0,"",0,"",0,"",0,"",0,"",0,"",0,"",0,"",0,0,0,0,0,0,0,0,0,0,0,0,0,0,0,0,0,0,0,0,0,0,0,0,0,0,0,0,0,0,0,0,0,0,0,0,0],FALSE],
    [[0,0,0,"",0,0,"",0,0,0,"",0,"",0,"",0,"",0,"",0,"",0,"",0,"",0,0,0,0,0,0,0,0,0,0,0,0,0,0,0,0,0,0,0,0,0,0,0,0,0,0,0,0,0,0,0,0,0,0,0,0,0],FALSE],
    [[0,0,0,"",0,0,"",0,0,0,"",0,"",0,"",0,"",0,"",0,"",0,"",0,"",0,0,0,0,0,0,0,0,0,0,0,0,0,0,0,0,0,0,0,0,0,0,0,0,0,0,0,0,0,0,0,0,0,0,0,0,0],FALSE],
    [[0,0,0,"",0,0,"",0,0,0,"",0,"",0,"",0,"",0,"",0,"",0,"",0,"",0,0,0,0,0,0,0,0,0,0,0,0,0,0,0,0,0,0,0,0,0,0,0,0,0,0,0,0,0,0,0,0,0,0,0,0,0],FALSE],
    [[0,0,0,"",0,0,"",0,0,0,"",0,"",0,"",0,"",0,"",0,"",0,"",0,"",0,0,0,0,0,0,0,0,0,0,0,0,0,0,0,0,0,0,0,0,0,0,0,0,0,0,0,0,0,0,0,0,0,0,0,0,0],FALSE]],

    [[[0,0,0,"",0,0,"",0,0,0,"",0,"",0,"",0,"",0,"",0,"",0,"",0,"",0,0,0,0,0,0,0,0,0,0,0,0,0,0,0,0,0,0,0,0,0,0,0,0,0,0,0,0,0,0,0,0,0,0,0,0,0],FALSE],
    [[0,0,0,"",0,0,"",0,0,0,"",0,"",0,"",0,"",0,"",0,"",0,"",0,"",0,0,0,0,0,0,0,0,0,0,0,0,0,0,0,0,0,0,0,0,0,0,0,0,0,0,0,0,0,0,0,0,0,0,0,0,0],FALSE],
    [[0,0,0,"",0,0,"",0,0,0,"",0,"",0,"",0,"",0,"",0,"",0,"",0,"",0,0,0,0,0,0,0,0,0,0,0,0,0,0,0,0,0,0,0,0,0,0,0,0,0,0,0,0,0,0,0,0,0,0,0,0,0],FALSE],
    [[0,0,0,"",0,0,"",0,0,0,"",0,"",0,"",0,"",0,"",0,"",0,"",0,"",0,0,0,0,0,0,0,0,0,0,0,0,0,0,0,0,0,0,0,0,0,0,0,0,0,0,0,0,0,0,0,0,0,0,0,0,0],FALSE],
    [[0,0,0,"",0,0,"",0,0,0,"",0,"",0,"",0,"",0,"",0,"",0,"",0,"",0,0,0,0,0,0,0,0,0,0,0,0,0,0,0,0,0,0,0,0,0,0,0,0,0,0,0,0,0,0,0,0,0,0,0,0,0],FALSE],
    [[0,0,0,"",0,0,"",0,0,0,"",0,"",0,"",0,"",0,"",0,"",0,"",0,"",0,0,0,0,0,0,0,0,0,0,0,0,0,0,0,0,0,0,0,0,0,0,0,0,0,0,0,0,0,0,0,0,0,0,0,0,0],FALSE],
    [[0,0,0,"",0,0,"",0,0,0,"",0,"",0,"",0,"",0,"",0,"",0,"",0,"",0,0,0,0,0,0,0,0,0,0,0,0,0,0,0,0,0,0,0,0,0,0,0,0,0,0,0,0,0,0,0,0,0,0,0,0,0],FALSE],
    [[0,0,0,"",0,0,"",0,0,0,"",0,"",0,"",0,"",0,"",0,"",0,"",0,"",0,0,0,0,0,0,0,0,0,0,0,0,0,0,0,0,0,0,0,0,0,0,0,0,0,0,0,0,0,0,0,0,0,0,0,0,0],FALSE],
    [[0,0,0,"",0,0,"",0,0,0,"",0,"",0,"",0,"",0,"",0,"",0,"",0,"",0,0,0,0,0,0,0,0,0,0,0,0,0,0,0,0,0,0,0,0,0,0,0,0,0,0,0,0,0,0,0,0,0,0,0,0,0],FALSE],
    [[0,0,0,"",0,0,"",0,0,0,"",0,"",0,"",0,"",0,"",0,"",0,"",0,"",0,0,0,0,0,0,0,0,0,0,0,0,0,0,0,0,0,0,0,0,0,0,0,0,0,0,0,0,0,0,0,0,0,0,0,0,0],FALSE]],

    [[[0,0,0,"",0,0,"",0,0,0,"",0,"",0,"",0,"",0,"",0,"",0,"",0,"",0,0,0,0,0,0,0,0,0,0,0,0,0,0,0,0,0,0,0,0,0,0,0,0,0,0,0,0,0,0,0,0,0,0,0,0,0],FALSE],
    [[0,0,0,"",0,0,"",0,0,0,"",0,"",0,"",0,"",0,"",0,"",0,"",0,"",0,0,0,0,0,0,0,0,0,0,0,0,0,0,0,0,0,0,0,0,0,0,0,0,0,0,0,0,0,0,0,0,0,0,0,0,0],FALSE],
    [[0,0,0,"",0,0,"",0,0,0,"",0,"",0,"",0,"",0,"",0,"",0,"",0,"",0,0,0,0,0,0,0,0,0,0,0,0,0,0,0,0,0,0,0,0,0,0,0,0,0,0,0,0,0,0,0,0,0,0,0,0,0],FALSE],
    [[0,0,0,"",0,0,"",0,0,0,"",0,"",0,"",0,"",0,"",0,"",0,"",0,"",0,0,0,0,0,0,0,0,0,0,0,0,0,0,0,0,0,0,0,0,0,0,0,0,0,0,0,0,0,0,0,0,0,0,0,0,0],FALSE],
    [[0,0,0,"",0,0,"",0,0,0,"",0,"",0,"",0,"",0,"",0,"",0,"",0,"",0,0,0,0,0,0,0,0,0,0,0,0,0,0,0,0,0,0,0,0,0,0,0,0,0,0,0,0,0,0,0,0,0,0,0,0,0],FALSE],
    [[0,0,0,"",0,0,"",0,0,0,"",0,"",0,"",0,"",0,"",0,"",0,"",0,"",0,0,0,0,0,0,0,0,0,0,0,0,0,0,0,0,0,0,0,0,0,0,0,0,0,0,0,0,0,0,0,0,0,0,0,0,0],FALSE],
    [[0,0,0,"",0,0,"",0,0,0,"",0,"",0,"",0,"",0,"",0,"",0,"",0,"",0,0,0,0,0,0,0,0,0,0,0,0,0,0,0,0,0,0,0,0,0,0,0,0,0,0,0,0,0,0,0,0,0,0,0,0,0],FALSE],
    [[0,0,0,"",0,0,"",0,0,0,"",0,"",0,"",0,"",0,"",0,"",0,"",0,"",0,0,0,0,0,0,0,0,0,0,0,0,0,0,0,0,0,0,0,0,0,0,0,0,0,0,0,0,0,0,0,0,0,0,0,0,0],FALSE],
    [[0,0,0,"",0,0,"",0,0,0,"",0,"",0,"",0,"",0,"",0,"",0,"",0,"",0,0,0,0,0,0,0,0,0,0,0,0,0,0,0,0,0,0,0,0,0,0,0,0,0,0,0,0,0,0,0,0,0,0,0,0,0],FALSE],
    [[0,0,0,"",0,0,"",0,0,0,"",0,"",0,"",0,"",0,"",0,"",0,"",0,"",0,0,0,0,0,0,0,0,0,0,0,0,0,0,0,0,0,0,0,0,0,0,0,0,0,0,0,0,0,0,0,0,0,0,0,0,0],FALSE]]];

ENDMODULE
